// TIA Portal project "Lift" (V15.1)

(* hardware
DEVICE "S7-1200 station_1"  S7-1200 Station
   slot 0: "Rack_0"  S7-1200 Rack  Rack  V1.0
   slot 1: "PLC_1"  CPU 1215C DC/DC/DC  6ES7 215-1AG40-0XB0  V4.2
*)

// ===== PLC "PLC_1"  CPU 1215C DC/DC/DC =====

VAR_GLOBAL   // PLC tag table "Default tag table"
   "Clock_Byte" AT %MB1 : Byte;
   "Clock_10Hz" AT %M1.0 : Bool;
   "Clock_5Hz" AT %M1.1 : Bool;
   "Clock_2.5Hz" AT %M1.2 : Bool;
   "Clock_2Hz" AT %M1.3 : Bool;
   "Clock_1.25Hz" AT %M1.4 : Bool;
   "Clock_1Hz" AT %M1.5 : Bool;
   "Clock_0.625Hz" AT %M1.6 : Bool;
   "Clock_0.5Hz" AT %M1.7 : Bool;
END_VAR

VAR_GLOBAL   // PLC tag table "lift butoane interior"
   "buton_parter" AT %I0.0 : Bool;
   "buton_et1" AT %I0.1 : Bool;
   "buton_et2" AT %I0.2 : Bool;
   "butor_urgenta" AT %I0.3 : Bool;
   "reset_button_urgenta" AT %I0.4 : Bool;
END_VAR

VAR_GLOBAL   // PLC tag table "lift outputs"
   "usa_parter" AT %Q0.0 : Bool;
   "usa_et1" AT %Q0.1 : Bool;
   "usa_et2" AT %Q0.2 : Bool;
   "bec_lift" AT %Q0.3 : Bool;
   "usa lift" AT %Q0.4 : Bool;
END_VAR

VAR_GLOBAL   // PLC tag table "lift auxiliares"
   "block_request_parter" AT %M0.0 : Bool;
   "urgenta_pressed" AT %M2.0 : Bool;
   "block_request_et1" AT %M2.1 : Bool;
   "block_request_et2" AT %M2.2 : Bool;
   "directie sus" AT %M2.3 : Bool;
   "directie jos" AT %M2.4 : Bool;
   "block_persoana" AT %M2.5 : Bool;
   "limitator_parter" AT %M2.6 : Bool;
   "limitator_1" AT %M2.7 : Bool;
   "limitator_2" AT %M3.0 : Bool;
END_VAR

VAR_GLOBAL   // PLC tag table "lift butoane exterior"
   "buton_exterior_parter" AT %I0.5 : Bool;
   "buton_et1_ext" AT %I0.6 : Bool;
   "buton_et2_ext" AT %I0.7 : Bool;
END_VAR

DATA_BLOCK "motor_DB"   // DB1
{ S7_Optimized_Access := 'TRUE' }
VERSION : 0.1
// stored: InstanceOfName motor parter
"motor parter"
BEGIN
END_DATA_BLOCK

DATA_BLOCK "motor_DB_1"   // DB2
{ S7_Optimized_Access := 'TRUE' }
VERSION : 0.1
// stored: InstanceOfName motor parter
"motor parter"
BEGIN
END_DATA_BLOCK

DATA_BLOCK "motor_DB_2"   // DB3
{ S7_Optimized_Access := 'TRUE' }
VERSION : 0.1
// stored: InstanceOfName motor parter
"motor parter"
BEGIN
END_DATA_BLOCK

DATA_BLOCK "motor et1_DB"   // DB4
{ S7_Optimized_Access := 'TRUE' }
VERSION : 0.1
// stored: InstanceOfName motor et1
"motor et1"
BEGIN
END_DATA_BLOCK

DATA_BLOCK "motor et2_DB"   // DB5
{ S7_Optimized_Access := 'TRUE' }
VERSION : 0.1
// stored: InstanceOfName motor et2
"motor et2"
BEGIN
END_DATA_BLOCK

FUNCTION_BLOCK "motor parter"   // FB1, LAD
{ S7_Optimized_Access := 'TRUE' }
VERSION : 0.1
   VAR_INPUT
      req_p : Bool;
      et_p : Bool;
      et_1 : Bool;
      et_2 : Bool;
   END_VAR
   VAR_OUTPUT
      dir_sus : Bool;
      dir_jos : Bool;
   END_VAR
BEGIN

REGION Network 1: cerere de la parter
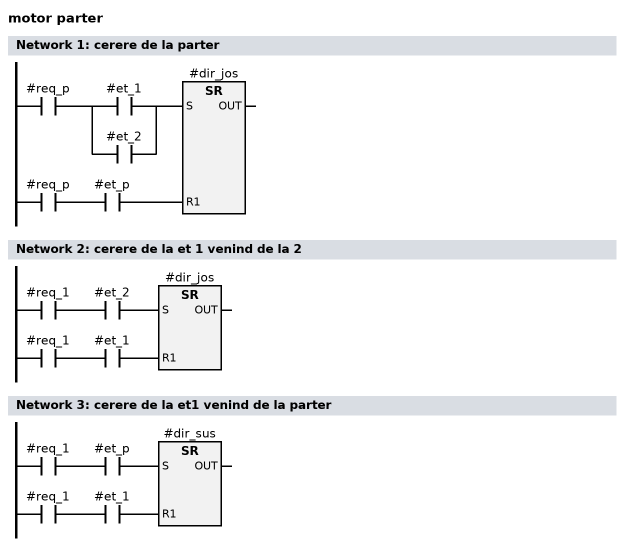
   RUNG wire#powerrail
      Contact( #req_p )
      wire#w1
      Contact( #et_1 )
      wire#w2
      S_SR(operand := #dir_jos, r1 := wire#w3)
   END_RUNG
   RUNG wire#w1
      Contact( #et_2 )
   END_RUNG wire#w2
   RUNG wire#powerrail
      Contact( #req_p )
      Contact( #et_p )
   END_RUNG wire#w3
   // the same network as SCL:
   IF #req_p AND (#et_1 OR #et_2) THEN
       #dir_jos := TRUE;   // SR flip-flop
   END_IF;
   IF #req_p AND #et_p THEN #dir_jos := FALSE; END_IF;
END_REGION

REGION Network 2: cerere de la et 1 venind de la 2
   RUNG wire#powerrail
      Contact( #req_1 )
      Contact( #et_2 )
      S_SR(operand := #dir_jos, r1 := wire#w1)
   END_RUNG
   RUNG wire#powerrail
      Contact( #req_1 )
      Contact( #et_1 )
   END_RUNG wire#w1
   // the same network as SCL:
   IF #req_1 AND #et_2 THEN
       #dir_jos := TRUE;   // SR flip-flop
   END_IF;
   IF #req_1 AND #et_1 THEN #dir_jos := FALSE; END_IF;
END_REGION

REGION Network 3: cerere de la et1 venind de la parter
   RUNG wire#powerrail
      Contact( #req_1 )
      Contact( #et_p )
      S_SR(operand := #dir_sus, r1 := wire#w1)
   END_RUNG
   RUNG wire#powerrail
      Contact( #req_1 )
      Contact( #et_1 )
   END_RUNG wire#w1
   // the same network as SCL:
   IF #req_1 AND #et_p THEN
       #dir_sus := TRUE;   // SR flip-flop
   END_IF;
   IF #req_1 AND #et_1 THEN #dir_sus := FALSE; END_IF;
END_REGION
END_FUNCTION_BLOCK

FUNCTION_BLOCK "motor et2"   // FB2, LAD
{ S7_Optimized_Access := 'TRUE' }
VERSION : 0.1
   VAR_INPUT
      req_2 : Bool;
      et_p : Bool;
      et_1 : Bool;
      et_2 : Bool;
   END_VAR
   VAR_OUTPUT
      dir_sus : Bool;
      dir_jos : Bool;
   END_VAR
BEGIN

REGION Network 1: cerere de la etaj 2
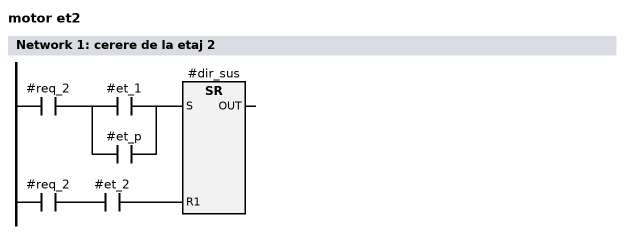
   RUNG wire#powerrail
      Contact( #req_2 )
      wire#w1
      Contact( #et_1 )
      wire#w2
      S_SR(operand := #dir_sus, r1 := wire#w3)
   END_RUNG
   RUNG wire#w1
      Contact( #et_p )
   END_RUNG wire#w2
   RUNG wire#powerrail
      Contact( #req_2 )
      Contact( #et_2 )
   END_RUNG wire#w3
   // the same network as SCL:
   IF #req_2 AND (#et_1 OR #et_p) THEN
       #dir_sus := TRUE;   // SR flip-flop
   END_IF;
   IF #req_2 AND #et_2 THEN #dir_sus := FALSE; END_IF;
END_REGION
END_FUNCTION_BLOCK

FUNCTION_BLOCK "motor et1"   // FB3, LAD
{ S7_Optimized_Access := 'TRUE' }
VERSION : 0.1
   VAR_INPUT
      req_1 : Bool;
      et_p : Bool;
      et_1 : Bool;
      et_2 : Bool;
   END_VAR
   VAR_OUTPUT
      dir_sus : Bool;
      dir_jos : Bool;
   END_VAR
BEGIN

REGION Network 1: cerere de la et 1 venind de la 2
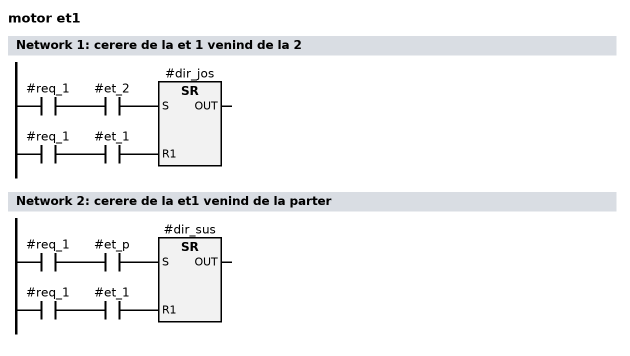
   RUNG wire#powerrail
      Contact( #req_1 )
      Contact( #et_2 )
      S_SR(operand := #dir_jos, r1 := wire#w1)
   END_RUNG
   RUNG wire#powerrail
      Contact( #req_1 )
      Contact( #et_1 )
   END_RUNG wire#w1
   // the same network as SCL:
   IF #req_1 AND #et_2 THEN
       #dir_jos := TRUE;   // SR flip-flop
   END_IF;
   IF #req_1 AND #et_1 THEN #dir_jos := FALSE; END_IF;
END_REGION

REGION Network 2: cerere de la et1 venind de la parter
   RUNG wire#powerrail
      Contact( #req_1 )
      Contact( #et_p )
      S_SR(operand := #dir_sus, r1 := wire#w1)
   END_RUNG
   RUNG wire#powerrail
      Contact( #req_1 )
      Contact( #et_1 )
   END_RUNG wire#w1
   // the same network as SCL:
   IF #req_1 AND #et_p THEN
       #dir_sus := TRUE;   // SR flip-flop
   END_IF;
   IF #req_1 AND #et_1 THEN #dir_sus := FALSE; END_IF;
END_REGION
END_FUNCTION_BLOCK

ORGANIZATION_BLOCK "Main"   // OB1, LAD, ProgramCycle
TITLE = "Main Program Sweep (Cycle)"
{ S7_Optimized_Access := 'TRUE' }
VERSION : 0.1
   VAR_INPUT
      Initial_Call : Bool;   // Initial call of this OB
      Remanence : Bool;   // =True, if remanent data are available
   END_VAR
   VAR_TEMP   // added for the SCL form of the ladder/FBD networks
      _w1 : Bool;
      _w2 : Bool;
      _w3 : Bool;
   END_VAR
BEGIN

REGION Network 1: lift butoane pe etaj(sa vina la etajul cerut)
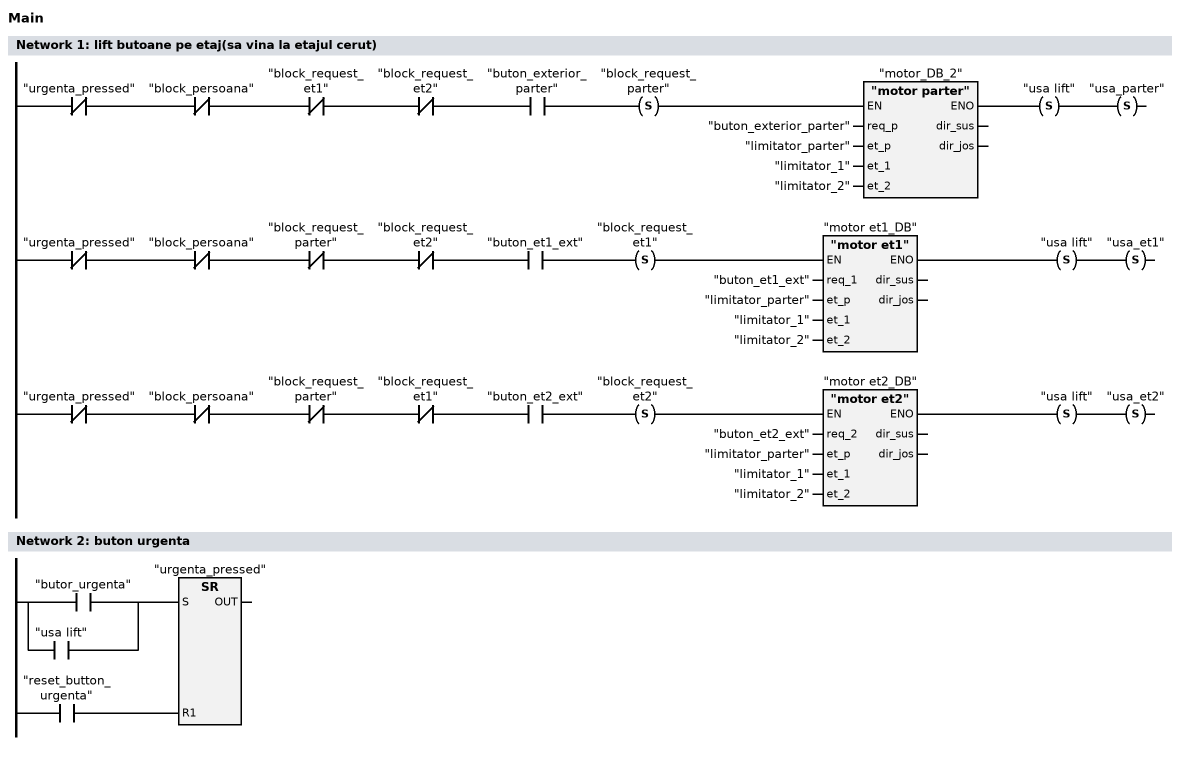
   RUNG wire#powerrail
      I_Contact( "urgenta_pressed" )
      I_Contact( "block_persoana" )
      I_Contact( "block_request_et1" )
      I_Contact( "block_request_et2" )
      Contact( "buton_exterior_parter" )
      S_Coil( "block_request_parter" )
      "motor_DB_2"(req_p := "buton_exterior_parter", et_p := "limitator_parter", et_1 := "limitator_1", et_2 := "limitator_2", dir_sus =>, dir_jos =>)
      S_Coil( "usa lift" )
      S_Coil( "usa_parter" )
   END_RUNG
   RUNG wire#powerrail
      I_Contact( "urgenta_pressed" )
      I_Contact( "block_persoana" )
      I_Contact( "block_request_parter" )
      I_Contact( "block_request_et2" )
      Contact( "buton_et1_ext" )
      S_Coil( "block_request_et1" )
      "motor et1_DB"(req_1 := "buton_et1_ext", et_p := "limitator_parter", et_1 := "limitator_1", et_2 := "limitator_2", dir_sus =>, dir_jos =>)
      S_Coil( "usa lift" )
      S_Coil( "usa_et1" )
   END_RUNG
   RUNG wire#powerrail
      I_Contact( "urgenta_pressed" )
      I_Contact( "block_persoana" )
      I_Contact( "block_request_parter" )
      I_Contact( "block_request_et1" )
      Contact( "buton_et2_ext" )
      S_Coil( "block_request_et2" )
      "motor et2_DB"(req_2 := "buton_et2_ext", et_p := "limitator_parter", et_1 := "limitator_1", et_2 := "limitator_2", dir_sus =>, dir_jos =>)
      S_Coil( "usa lift" )
      S_Coil( "usa_et2" )
   END_RUNG
   // the same network as SCL:
   IF NOT "urgenta_pressed" AND NOT "block_persoana" AND NOT "block_request_et1" AND NOT "block_request_et2" AND "buton_exterior_parter" THEN
       "block_request_parter" := TRUE;
   END_IF;
   "motor_DB_2"(EN := NOT "urgenta_pressed" AND NOT "block_persoana" AND NOT "block_request_et1" AND NOT "block_request_et2" AND "buton_exterior_parter",   // "motor parter"
                req_p := "buton_exterior_parter",
                et_p := "limitator_parter",
                et_1 := "limitator_1",
                et_2 := "limitator_2",
                ENO => #_w1);
   IF #_w1 THEN
       "usa lift" := TRUE;
       "usa_parter" := TRUE;
   END_IF;
   IF NOT "urgenta_pressed" AND NOT "block_persoana" AND NOT "block_request_parter" AND NOT "block_request_et2" AND "buton_et1_ext" THEN
       "block_request_et1" := TRUE;
   END_IF;
   "motor et1_DB"(EN := NOT "urgenta_pressed" AND NOT "block_persoana" AND NOT "block_request_parter" AND NOT "block_request_et2" AND "buton_et1_ext",   // "motor et1"
                  req_1 := "buton_et1_ext",
                  et_p := "limitator_parter",
                  et_1 := "limitator_1",
                  et_2 := "limitator_2",
                  ENO => #_w2);
   IF #_w2 THEN
       "usa lift" := TRUE;
       "usa_et1" := TRUE;
   END_IF;
   IF NOT "urgenta_pressed" AND NOT "block_persoana" AND NOT "block_request_parter" AND NOT "block_request_et1" AND "buton_et2_ext" THEN
       "block_request_et2" := TRUE;
   END_IF;
   "motor et2_DB"(EN := NOT "urgenta_pressed" AND NOT "block_persoana" AND NOT "block_request_parter" AND NOT "block_request_et1" AND "buton_et2_ext",   // "motor et2"
                  req_2 := "buton_et2_ext",
                  et_p := "limitator_parter",
                  et_1 := "limitator_1",
                  et_2 := "limitator_2",
                  ENO => #_w3);
   IF #_w3 THEN
       "usa lift" := TRUE;
       "usa_et2" := TRUE;
   END_IF;
END_REGION

REGION Network 2: buton urgenta
   RUNG wire#powerrail
      Contact( "butor_urgenta" )
      wire#w1
      S_SR(operand := "urgenta_pressed", r1 := wire#w2)
   END_RUNG
   RUNG wire#powerrail
      Contact( "usa lift" )
   END_RUNG wire#w1
   RUNG wire#powerrail
      Contact( "reset_button_urgenta" )
   END_RUNG wire#w2
   // the same network as SCL:
   IF "butor_urgenta" OR "usa lift" THEN
       "urgenta_pressed" := TRUE;   // SR flip-flop
   END_IF;
   IF "reset_button_urgenta" THEN "urgenta_pressed" := FALSE; END_IF;
END_REGION

REGION Network 3: urcare la etajul cerut
END_REGION
END_ORGANIZATION_BLOCK